INTERFACE I_DINT EXTENDS I_Datatype

PROPERTY PUBLIC Value : REFERENCE TO DINT
GET
END_GET
END_PROPERTY

END_INTERFACE

(* stored: Version 1.1.0.1, ProductVersion 3.1.4024.15
   Itf I_DINT: Id {98ffdff1-1a46-099d-2567-8d2a1f656e58}
   Property Value: Id {1afc3a72-cc3c-00c6-057f-98a4091f8af1}
   Get Get: Id {ad3e71ca-7d9d-0db7-2066-470b341ce68d} *)
